RESOURCE_TYPE _Core0
  (* Standard: 61499-2 *)
  (* Version 0.1, 2017-00-09, hpea485, UOA *)
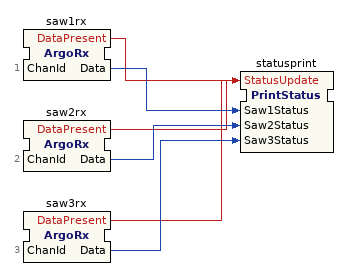
  FBS
    saw1rx : ArgoRx(ChanId := 1);
    saw2rx : ArgoRx(ChanId := 2);
    saw3rx : ArgoRx(ChanId := 3);
    statusprint : PrintStatus;
  END_FBS
  EVENT_CONNECTIONS
    saw1rx.DataPresent TO statusprint.StatusUpdate;
    saw2rx.DataPresent TO statusprint.StatusUpdate;
    saw3rx.DataPresent TO statusprint.StatusUpdate;
  END_CONNECTIONS
  DATA_CONNECTIONS
    saw1rx.Data TO statusprint.Saw1Status;
    saw2rx.Data TO statusprint.Saw2Status;
    saw3rx.Data TO statusprint.Saw3Status;
  END_CONNECTIONS
END_RESOURCE_TYPE
